FUNCTION_BLOCK POU IMPLEMENTS ITcTask
VAR_INPUT
END_VAR
VAR_OUTPUT
END_VAR
VAR
END_VAR

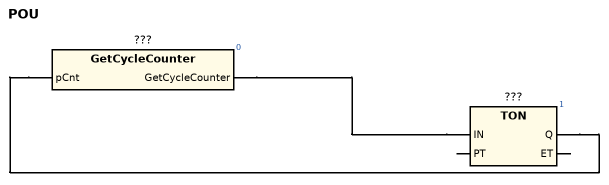
???(pCnt := ???.Q); // GetCycleCounter
???(IN := ???.GetCycleCounter); // TON

{attribute 'TcTypeSystem'}
{attribute 'no-analysis'}
{attribute 'c++_compatible'}
{attribute 'minimal_input_size' := '4'}
{attribute 'pack_mode' := '4'}
{warning 'add method implementation '}
METHOD GetCurrentDcTime : HRESULT
VAR_INPUT
	pDcTime	: POINTER TO UDINT;
END_VAR
END_METHOD

{attribute 'TcTypeSystem'}
{attribute 'no-analysis'}
{attribute 'c++_compatible'}
{attribute 'minimal_input_size' := '4'}
{attribute 'pack_mode' := '4'}
{warning 'add method implementation '}
METHOD GetCurrentSysTime : HRESULT
VAR_INPUT
	pSysTime	: POINTER TO ULINT;
END_VAR
END_METHOD

{attribute 'TcTypeSystem'}
{attribute 'no-analysis'}
{attribute 'c++_compatible'}
{attribute 'minimal_input_size' := '4'}
{attribute 'pack_mode' := '4'}
{warning 'add method implementation '}
METHOD GetCycleCounter : HRESULT
VAR_INPUT
	pCnt	: POINTER TO ULINT;
END_VAR
END_METHOD

{attribute 'TcTypeSystem'}
{attribute 'no-analysis'}
{attribute 'c++_compatible'}
{attribute 'minimal_input_size' := '4'}
{attribute 'pack_mode' := '4'}
{warning 'add method implementation '}
METHOD GetCycleTime : HRESULT
VAR_INPUT
	pCycleTimeNS	: POINTER TO UDINT;
END_VAR
END_METHOD

{attribute 'TcTypeSystem'}
{attribute 'no-analysis'}
{attribute 'c++_compatible'}
{attribute 'minimal_input_size' := '4'}
{attribute 'pack_mode' := '4'}
{warning 'add method implementation '}
METHOD GetPriority : HRESULT
VAR_INPUT
	pPriority	: POINTER TO UDINT;
END_VAR
END_METHOD

{attribute 'TcTypeSystem'}
{attribute 'no-analysis'}
{attribute 'c++_compatible'}
{attribute 'minimal_input_size' := '4'}
{attribute 'pack_mode' := '4'}
{warning 'add method implementation '}
METHOD TcAddRef : UDINT
END_METHOD

{attribute 'TcTypeSystem'}
{attribute 'no-analysis'}
{attribute 'c++_compatible'}
{attribute 'minimal_input_size' := '4'}
{attribute 'pack_mode' := '4'}
{warning 'add method implementation '}
METHOD TcQueryInterface : HRESULT
VAR_INPUT
	iid	: REFERENCE TO IID;
	pipItf	: POINTER TO PVOID;
END_VAR
END_METHOD

{attribute 'TcTypeSystem'}
{attribute 'no-analysis'}
{attribute 'c++_compatible'}
{attribute 'minimal_input_size' := '4'}
{attribute 'pack_mode' := '4'}
{warning 'add method implementation '}
METHOD TcRelease : UDINT
END_METHOD

END_FUNCTION_BLOCK

(* stored: Version 1.1.0.1, ProductVersion 3.1.4024.4
   POU POU: Id {63d1d78c-7b37-4193-975a-102534b592d4}, SpecialFunc None
   Method GetCurrentDcTime: Id {e23d95f0-309c-4d99-b87e-7fb476b40564}
   Method GetCurrentSysTime: Id {918272e7-aeca-4b50-b5f3-7af73d594efc}
   Method GetCycleCounter: Id {dd694eaf-e961-4030-bd43-a8223e510f93}
   Method GetCycleTime: Id {41f45920-515a-4f8d-ba5b-b2803aa5c303}
   Method GetPriority: Id {0c307687-172f-4a7f-9c96-59de1d4fa317}
   Method TcAddRef: Id {c1641772-bcc9-4331-bd4d-2377671af6d4}
   Method TcQueryInterface: Id {e423decd-03c6-4d63-b3a8-90b50c9ec30c}
   Method TcRelease: Id {0844a398-2965-4c20-9f97-92947e23057b} *)
